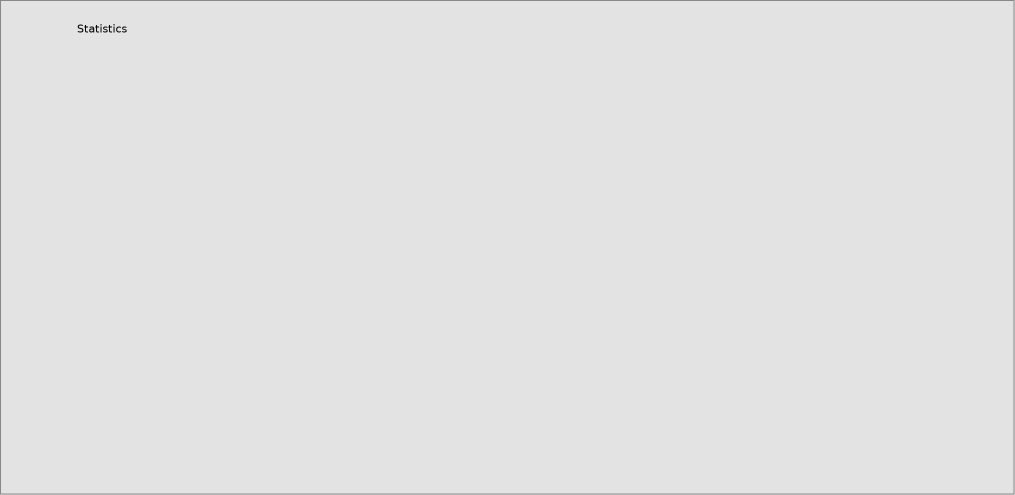
VISUALIZATION F_05_Statistics  // 1015x495
VAR_IN_OUT
	stScreenData	: ST_MCHMIPrepareScreen_05_XX;
	
END_VAR
    Label (27,14 150x30), "Statistics"
END_VISUALIZATION

(* stored: Version 1.1.0.1
   Visu F_05_Statistics: Id {d2a844fd-5f20-0b85-1f04-c107406010af} *)
